FUNCTION_BLOCK ScriblySequenceGoHome EXTENDS ScriblySequence IMPLEMENTS ZCore.ISequence
VAR
  _step : ZCore.Step(ScriblyStep.GohomeBegin, ScriblyStep.GohomeEnd);
  _timer : ZAux.Timer;
END_VAR

IF NOT Busy THEN
  RETURN;
END_IF

IF OnStart(_step) THEN
  ; // init custom sequence variables here ...
END_IF

IF OnStop() THEN
  RETURN; // external stop was triggered
END_IF

IF OnHalt() THEN
  ; // Halting := TRUE; // Uncomment to acknowledge that the sequence is halting
END_IF

REPEAT
  LogStep();

  CASE _step.Index OF
    (* -------------------------------------------------------------------------------------------------------------------------------- *)
    ScriblyStep.GoHomeBegin:
    (* -------------------------------------------------------------------------------------------------------------------------------- *)
      IF _step.OnEntry()
      THEN
        ;
			END_IF

      _step.SetNext(index:=ScriblyStep.GoHomeMoveUp);

    (* -------------------------------------------------------------------------------------------------------------------------------- *)
    ScriblyStep.GoHomeMoveUp:
    (* -------------------------------------------------------------------------------------------------------------------------------- *)
      IF _step.OnEntry()
      THEN
        _actuator.Pen.UpAsync(THIS^);
        _axis.AxisX.StopAsync(THIS^);
        _axis.AxisY.StopAsync(THIS^);
			END_IF
      
      Await(_actuator.Pen, nextStep:=ScriblyStep.GoHomeReferenceXY);

    (* -------------------------------------------------------------------------------------------------------------------------------- *)
    ScriblyStep.GoHomeReferenceXY:
    (* -------------------------------------------------------------------------------------------------------------------------------- *)
      IF _step.OnEntry()
      THEN
        _axis.AxisX.HomingAsync(THIS^);
        _axis.AxisY.HomingAsync(THIS^);
			END_IF
      
      Await3(_actuator.Pen, _axis.AxisX, _axis.AxisY, nextStep:=ScriblyStep.GoHomeEnd);

    (* -------------------------------------------------------------------------------------------------------------------------------- *)
    ScriblyStep.GoHomeEnd:
    (* -------------------------------------------------------------------------------------------------------------------------------- *)
      SetBusy(FALSE);
  
  ELSE
    Abort('sequence contains unhandled step');
  END_CASE
UNTIL _step.IsNotRepeatable() OR_ELSE NOT Busy END_REPEAT

END_FUNCTION_BLOCK

(* stored: Version 1.1.0.1
   POU ScriblySequenceGoHome: Id {b9e68848-6e34-449f-85c9-c7a943e2fd10}, SpecialFunc None *)
